Omron CX-Programmer project NewProject (CX-Programmer 9.73)

# PLC NewPLC1: CP1E N20

## Global symbols (name address type ; comment)
0.00 BOOL  ; sensor
100.07 BOOL  ; lamp 1
C001 BOOL  ; counter
T001 BOOL  ; timer

## Program NewProgram1 (cyclic task 0)

### Section Section1

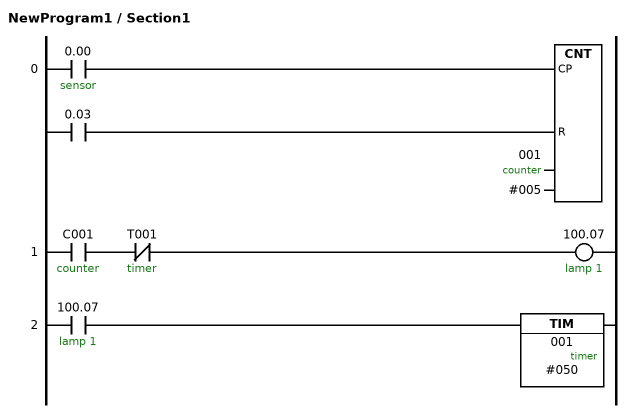
; rung 0
LD 0.00  ; sensor
LD 0.03
CNT 001 #005  ; counter
; rung 1
LD C001  ; counter
ANDNOT T001  ; timer
OUT 100.07  ; lamp 1
; rung 2
LD 100.07  ; lamp 1
TIM 001 #050  ; timer

### Section END
; rung 0
END(001)